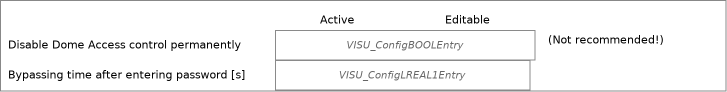
VISUALIZATION VISU_SafetyConfig_DomeAccessGeneral  // 727x92
VAR_IN_OUT
    editable : SafetyDomeAccessConfig;
	active : SafetyDomeAccessConfig;
END_VAR
    Frame (275,30 260x30), tooltip "The number of steps which should be carried out at minimum to counter-act the backlash in the system during the final move (for Z axis: at low speed)"
        shows VISU_ConfigBOOLEntry(active := active.disabled, editable := editable.disabled)
    Label (275,10 125x20), "Active"
    Label (405,10 125x20), "Editable"
    Label (5,60 250x30), "Bypassing time after entering password [s]"
    Frame (275,60 255x30), tooltip "The number of steps to be expected between the time at which the PLC realizes that the brake signal must be set, and the time that the axis is fully stopped (for Z axis: at low speed)"
        shows VISU_ConfigLREAL1Entry(active := active.bypassTimeAfterPassword, editable := editable.bypassTimeAfterPassword)
    Label (5,30 285x30), "Disable Dome Access control permanently"
    Label (545,25 180x30), "(Not recommended!)"
END_VISUALIZATION

(* stored: Version 1.1.0.1, ProductVersion 3.1.4019.2
   Visu VISU_SafetyConfig_DomeAccessGeneral: Id {8a228830-48b8-4881-a6a0-08514feea180} *)
